(* CODESYS project TrigaPLC.project
   Title: TrigaPLC
   Author: Thalles Campagnani
   Version: 0.0.1

Project tree, tasks and I/O mapping:
  TrigaPLC : TM251MESE, Schneider Electric, order no. TM251MESE, version 4.0.6.18
      settings: OPCUA enable = True; Dummy int param for online change = 28
    application Application
      libraries: Toolbox, 2.2.0.0 (Schneider Electric); SysTimeRtc, 3.5.1.0 (System); SysTimeCore, 3.4.1.20 (System); Standard64, * (System)
      task MAST (cyclic, interval 20 ms, priority 15, watchdog 100 ms x 1) calls _001_Geral_DateAndHour
      global variables GVL
      data type Manegement
      global variables PersistentVars
      OPCUASymbolConfiguration
      data type User
      data type Group
      Symbols
      program _001_Geral_DateAndHour [CFC]
      DataLogManager
        LogFile
      trace Trace (task MAST): 
    Serial_Line_1 : Serial line, Schneider Electric, version 4.0.6.18
    Ethernet_1 : Ethernet Network, Schneider Electric, version 4.0.6.18
        settings: IPAddress = [192, 168, 1, 1]; SubnetMask = [255, 255, 255, 0]; DeviceName = 'TrigaPLC'; WebServer = TRUE; FTP Server = TRUE; SoMachine Protocol = TRUE; Modbus Server = TRUE; NetManage Protocol = TRUE; SNMP protocol = TRUE; Enable Routing = FALSE; WebVisu protocol = TRUE
    COM_Bus : COM bus, Schneider Electric, version 4.0.6.18
    IO_Bus : IO bus - TM3, Schneider Electric, version 4.0.6.18
      Module_A2 : TM3AI8/G, Schneider Electric, order no. TM3AI8/G, version 1.0.0.17
          settings: KPI Configuration.KPI Configuration[0] = 32; KPI Configuration.KPI Configuration[1] = 32; KPI Configuration.KPI Configuration[2] = 32; KPI Configuration.KPI Configuration[3] = 32; KPI Configuration.KPI Configuration[4] = 32; KPI Configuration.KPI Configuration[5] = 32; KPI Configuration.KPI Configuration[6] = 32; KPI Configuration.KPI Configuration[7] = 32; KPI Configuration.KPI Configuration[9] = 0; KPI Configuration.KPI Configuration[11] = 0; KPI Configuration.KPI Configuration[13] = 0; KPI Configuration.KPI Configuration[15] = 0; KPI Configuration.KPI Configuration[17] = 0; KPI Configuration.KPI Configuration[19] = 0; KPI Configuration.KPI Configuration[21] = 0; KPI Configuration.KPI Configuration[23] = 0; KPI Configuration.KPI Configuration[24] = 0; KPI Configuration.KPI Configuration[25] = 32; KPI Configuration.KPI Configuration[26] = 0; KPI Configuration.KPI Configuration[27] = 32; KPI Configuration.KPI Configuration[28] = 0; KPI Configuration.KPI Configuration[29] = 32; KPI Configuration.KPI Configuration[30] = 0; KPI Configuration.KPI Configuration[31] = 32; KPI Configuration.KPI Configuration[32] = 0; KPI Configuration.KPI Configuration[33] = 32; KPI Configuration.KPI Configuration[34] = 0; KPI Configuration.KPI Configuration[35] = 32; KPI Configuration.KPI Configuration[36] = 0; KPI Configuration.KPI Configuration[37] = 32; KPI Configuration.KPI Configuration[38] = 0; KPI Configuration.KPI Configuration[39] = 32; KPI Configuration.KPI Configuration[40] = 2; KPI Configuration.KPI Configuration[42] = 2; KPI Configuration.KPI Configuration[44] = 2; KPI Configuration.KPI Configuration[46] = 2; KPI Configuration.KPI Configuration[48] = 2; KPI Configuration.KPI Configuration[50] = 2; KPI Configuration.KPI Configuration[52] = 2; KPI Configuration.KPI Configuration[54] = 2
          input  inSRadAre : INT  // IW0
          input  inSRadEntPri : INT  // IW1
          input  inSRadPoc : INT  // IW2
          input  inSRadRes : INT  // IW3
          input  inSRadSaiSec : INT  // IW4
          input  inSRadAer : INT  // IW5
          input  inReserva_AI26 : INT  // IW6
          input  inReserva_AI27 : INT  // IW7
          input  ibModule_12_IBStatusIW0 : BYTE  // IBStatusIW0
          input  ibModule_12_IBStatusIW1 : BYTE  // IBStatusIW1
          input  ibModule_12_IBStatusIW2 : BYTE  // IBStatusIW2
          input  ibModule_12_IBStatusIW3 : BYTE  // IBStatusIW3
          input  ibModule_12_IBStatusIW4 : BYTE  // IBStatusIW4
          input  ibModule_12_IBStatusIW5 : BYTE  // IBStatusIW5
          input  ibModule_12_IBStatusIW6 : BYTE  // IBStatusIW6
          input  ibModule_12_IBStatusIW7 : BYTE  // IBStatusIW7
      Module_A1 : TM3AI8/G, Schneider Electric, order no. TM3AI8/G, version 1.0.0.17
          settings: KPI Configuration.KPI Configuration[0] = 32; KPI Configuration.KPI Configuration[1] = 33; KPI Configuration.KPI Configuration[2] = 32; KPI Configuration.KPI Configuration[3] = 32; KPI Configuration.KPI Configuration[4] = 32; KPI Configuration.KPI Configuration[5] = 32; KPI Configuration.KPI Configuration[6] = 32; KPI Configuration.KPI Configuration[7] = 32; KPI Configuration.KPI Configuration[9] = 0; KPI Configuration.KPI Configuration[11] = 0; KPI Configuration.KPI Configuration[13] = 0; KPI Configuration.KPI Configuration[15] = 0; KPI Configuration.KPI Configuration[17] = 0; KPI Configuration.KPI Configuration[19] = 0; KPI Configuration.KPI Configuration[21] = 0; KPI Configuration.KPI Configuration[23] = 0; KPI Configuration.KPI Configuration[24] = 0; KPI Configuration.KPI Configuration[25] = 32; KPI Configuration.KPI Configuration[26] = 0; KPI Configuration.KPI Configuration[27] = 32; KPI Configuration.KPI Configuration[28] = 0; KPI Configuration.KPI Configuration[29] = 32; KPI Configuration.KPI Configuration[30] = 0; KPI Configuration.KPI Configuration[31] = 32; KPI Configuration.KPI Configuration[32] = 0; KPI Configuration.KPI Configuration[33] = 32; KPI Configuration.KPI Configuration[34] = 0; KPI Configuration.KPI Configuration[35] = 32; KPI Configuration.KPI Configuration[36] = 0; KPI Configuration.KPI Configuration[37] = 32; KPI Configuration.KPI Configuration[38] = 0; KPI Configuration.KPI Configuration[39] = 32; KPI Configuration.KPI Configuration[40] = 2; KPI Configuration.KPI Configuration[44] = 2; KPI Configuration.KPI Configuration[46] = 2; KPI Configuration.KPI Configuration[48] = 2; KPI Configuration.KPI Configuration[50] = 2; KPI Configuration.KPI Configuration[52] = 100; KPI Configuration.KPI Configuration[54] = 2
          input  inCPer : INT  // IW0
          input  inCLogARea : INT  // IW1
          input  inCLogALin : INT  // IW2
          input  inCLogALog : INT  // IW3
          input  inCLogAPer : INT  // IW4
          input  inCParALin : INT  // IW5
          input  inCParALog : INT  // IW6
          input  inCParAPer : INT  // IW7
          input  ibModule_11_IBStatusIW0 : BYTE  // IBStatusIW0
          input  ibModule_11_IBStatusIW1 : BYTE  // IBStatusIW1
          input  ibModule_11_IBStatusIW2 : BYTE  // IBStatusIW2
          input  ibModule_11_IBStatusIW3 : BYTE  // IBStatusIW3
          input  ibModule_11_IBStatusIW4 : BYTE  // IBStatusIW4
          input  ibModule_11_IBStatusIW5 : BYTE  // IBStatusIW5
          input  ibModule_11_IBStatusIW6 : BYTE  // IBStatusIW6
          input  ibModule_11_IBStatusIW7 : BYTE  // IBStatusIW7
      Module_A0 : TM3AI8/G, Schneider Electric, order no. TM3AI8/G, version 1.0.0.17
          settings: KPI Configuration.KPI Configuration[0] = 35; KPI Configuration.KPI Configuration[1] = 35; KPI Configuration.KPI Configuration[2] = 35; KPI Configuration.KPI Configuration[3] = 35; KPI Configuration.KPI Configuration[4] = 32; KPI Configuration.KPI Configuration[5] = 32; KPI Configuration.KPI Configuration[6] = 32; KPI Configuration.KPI Configuration[7] = 32; KPI Configuration.KPI Configuration[9] = 0; KPI Configuration.KPI Configuration[11] = 0; KPI Configuration.KPI Configuration[13] = 0; KPI Configuration.KPI Configuration[15] = 0; KPI Configuration.KPI Configuration[17] = 0; KPI Configuration.KPI Configuration[19] = 0; KPI Configuration.KPI Configuration[21] = 0; KPI Configuration.KPI Configuration[23] = 0; KPI Configuration.KPI Configuration[32] = 0; KPI Configuration.KPI Configuration[33] = 32; KPI Configuration.KPI Configuration[34] = 0; KPI Configuration.KPI Configuration[35] = 32; KPI Configuration.KPI Configuration[36] = 0; KPI Configuration.KPI Configuration[37] = 32; KPI Configuration.KPI Configuration[38] = 0; KPI Configuration.KPI Configuration[39] = 32; KPI Configuration.KPI Configuration[48] = 20; KPI Configuration.KPI Configuration[50] = 20; KPI Configuration.KPI Configuration[52] = 20
          input  inReserva_AI00 : INT  // IW0
          input  inReserva_AI01 : INT  // IW1
          input  inReserva_AI02 : INT  // IW2
          input  inReserva_AI03 : INT  // IW3
          input  inBarraReg : INT  // IW4
          input  inBarraCon : INT  // IW5
          input  inBarraSeg : INT  // IW6
          input  inCLin : INT  // IW7
          input  ibModule_13_IBStatusIW0 : BYTE  // IBStatusIW0
          input  ibModule_13_IBStatusIW1 : BYTE  // IBStatusIW1
          input  ibModule_13_IBStatusIW2 : BYTE  // IBStatusIW2
          input  ibModule_13_IBStatusIW3 : BYTE  // IBStatusIW3
          input  ibModule_13_IBStatusIW4 : BYTE  // IBStatusIW4
          input  ibModule_13_IBStatusIW5 : BYTE  // IBStatusIW5
          input  ibModule_13_IBStatusIW6 : BYTE  // IBStatusIW6
          input  ibModule_13_IBStatusIW7 : BYTE  // IBStatusIW7
      Module_A3 : TM3AI8/G, Schneider Electric, order no. TM3AI8/G, version 1.0.0.17
          settings: KPI Configuration.KPI Configuration[0] = 32; KPI Configuration.KPI Configuration[1] = 32; KPI Configuration.KPI Configuration[2] = 32; KPI Configuration.KPI Configuration[3] = 32; KPI Configuration.KPI Configuration[4] = 32; KPI Configuration.KPI Configuration[5] = 32; KPI Configuration.KPI Configuration[6] = 32; KPI Configuration.KPI Configuration[7] = 32; KPI Configuration.KPI Configuration[9] = 0; KPI Configuration.KPI Configuration[11] = 0; KPI Configuration.KPI Configuration[13] = 0; KPI Configuration.KPI Configuration[15] = 0; KPI Configuration.KPI Configuration[17] = 0; KPI Configuration.KPI Configuration[19] = 0; KPI Configuration.KPI Configuration[21] = 0; KPI Configuration.KPI Configuration[23] = 0; KPI Configuration.KPI Configuration[24] = 0; KPI Configuration.KPI Configuration[25] = 32; KPI Configuration.KPI Configuration[26] = 0; KPI Configuration.KPI Configuration[27] = 32; KPI Configuration.KPI Configuration[28] = 0; KPI Configuration.KPI Configuration[29] = 32; KPI Configuration.KPI Configuration[30] = 0; KPI Configuration.KPI Configuration[31] = 32; KPI Configuration.KPI Configuration[32] = 0; KPI Configuration.KPI Configuration[33] = 32; KPI Configuration.KPI Configuration[34] = 0; KPI Configuration.KPI Configuration[35] = 32; KPI Configuration.KPI Configuration[36] = 0; KPI Configuration.KPI Configuration[37] = 32; KPI Configuration.KPI Configuration[38] = 0; KPI Configuration.KPI Configuration[39] = 32; KPI Configuration.KPI Configuration[40] = 2; KPI Configuration.KPI Configuration[42] = 2; KPI Configuration.KPI Configuration[44] = 2; KPI Configuration.KPI Configuration[46] = 2; KPI Configuration.KPI Configuration[48] = 2; KPI Configuration.KPI Configuration[50] = 2; KPI Configuration.KPI Configuration[52] = 2; KPI Configuration.KPI Configuration[54] = 2
          input  inReserva_AI30 : INT  // IW0
          input  inReserva_AI31 : INT  // IW1
          input  inReserva_AI32 : INT  // IW2
          input  inReserva_AI33 : INT  // IW3
          input  inReserva_AI34 : INT  // IW4
          input  inReserva_AI35 : INT  // IW5
          input  inReserva_AI36 : INT  // IW6
          input  inReserva_AI37 : INT  // IW7
          input  ibModule_1_IBStatusIW0 : BYTE  // IBStatusIW0
          input  ibModule_1_IBStatusIW1 : BYTE  // IBStatusIW1
          input  ibModule_1_IBStatusIW2 : BYTE  // IBStatusIW2
          input  ibModule_1_IBStatusIW3 : BYTE  // IBStatusIW3
          input  ibModule_1_IBStatusIW4 : BYTE  // IBStatusIW4
          input  ibModule_1_IBStatusIW5 : BYTE  // IBStatusIW5
          input  ibModule_1_IBStatusIW6 : BYTE  // IBStatusIW6
          input  ibModule_1_IBStatusIW7 : BYTE  // IBStatusIW7
      Module_A4 : TM3AI8/G, Schneider Electric, order no. TM3AI8/G, version 1.0.0.17
          settings: KPI Configuration.KPI Configuration[0] = 35; KPI Configuration.KPI Configuration[1] = 35; KPI Configuration.KPI Configuration[2] = 35; KPI Configuration.KPI Configuration[3] = 35; KPI Configuration.KPI Configuration[4] = 35; KPI Configuration.KPI Configuration[5] = 35; KPI Configuration.KPI Configuration[6] = 35; KPI Configuration.KPI Configuration[7] = 35; KPI Configuration.KPI Configuration[9] = 0; KPI Configuration.KPI Configuration[11] = 0; KPI Configuration.KPI Configuration[13] = 0; KPI Configuration.KPI Configuration[15] = 0; KPI Configuration.KPI Configuration[17] = 0; KPI Configuration.KPI Configuration[19] = 0; KPI Configuration.KPI Configuration[21] = 0; KPI Configuration.KPI Configuration[23] = 0; KPI Configuration.KPI Configuration[24] = 0; KPI Configuration.KPI Configuration[25] = 32; KPI Configuration.KPI Configuration[26] = 0; KPI Configuration.KPI Configuration[27] = 32; KPI Configuration.KPI Configuration[28] = 0; KPI Configuration.KPI Configuration[29] = 32; KPI Configuration.KPI Configuration[30] = 0; KPI Configuration.KPI Configuration[31] = 32; KPI Configuration.KPI Configuration[32] = 0; KPI Configuration.KPI Configuration[33] = 32; KPI Configuration.KPI Configuration[34] = 0; KPI Configuration.KPI Configuration[35] = 32; KPI Configuration.KPI Configuration[36] = 0; KPI Configuration.KPI Configuration[37] = 32; KPI Configuration.KPI Configuration[38] = 0; KPI Configuration.KPI Configuration[39] = 32; KPI Configuration.KPI Configuration[40] = 2; KPI Configuration.KPI Configuration[42] = 2; KPI Configuration.KPI Configuration[44] = 2; KPI Configuration.KPI Configuration[46] = 2; KPI Configuration.KPI Configuration[48] = 2; KPI Configuration.KPI Configuration[50] = 2; KPI Configuration.KPI Configuration[52] = 2; KPI Configuration.KPI Configuration[54] = 2
          input  inSVasPri : INT  // IW0
          input  inReserva_AI41 : INT  // IW1
          input  inReserva_AI42 : INT  // IW2
          input  inReserva_AI43 : INT  // IW3
          input  inReserva_AI44 : INT  // IW4
          input  inReserva_AI45 : INT  // IW5
          input  inReserva_AI46 : INT  // IW6
          input  inReserva_AI47 : INT  // IW7
          input  ibModule_2_IBStatusIW0 : BYTE  // IBStatusIW0
          input  ibModule_2_IBStatusIW1 : BYTE  // IBStatusIW1
          input  ibModule_2_IBStatusIW2 : BYTE  // IBStatusIW2
          input  ibModule_2_IBStatusIW3 : BYTE  // IBStatusIW3
          input  ibModule_2_IBStatusIW4 : BYTE  // IBStatusIW4
          input  ibModule_2_IBStatusIW5 : BYTE  // IBStatusIW5
          input  ibModule_2_IBStatusIW6 : BYTE  // IBStatusIW6
          input  ibModule_2_IBStatusIW7 : BYTE  // IBStatusIW7
      Module_D0 : TM3DI16/G, Schneider Electric, order no. TM3DI16/G, version 1.0.1.4
          input  inModule_D0 : WORD  // IW0
          input  inCLinBit0 : BOOL  // IW0.I0
          input  inCLinBit1 : BOOL  // IW0.I1
          input  inCLinBit2 : BOOL  // IW0.I2
          input  inReserva_DI03 : BOOL  // IW0.I3
          input  inReserva_DI04 : BOOL  // IW0.I4
          input  inReserva_DI05 : BOOL  // IW0.I5
          input  inReserva_DI06 : BOOL  // IW0.I6
          input  inReserva_DI07 : BOOL  // IW0.I7
          input  inReserva_DI08 : BOOL  // IW0.I8
          input  inReserva_DI09 : BOOL  // IW0.I9
          input  inReserva_DI010 : BOOL  // IW0.I10
          input  inReserva_DI011 : BOOL  // IW0.I11
          input  inReserva_DI012 : BOOL  // IW0.I12
          input  inReserva_DI013 : BOOL  // IW0.I13
          input  inReserva_DI014 : BOOL  // IW0.I14
          input  inReserva_DI015 : BOOL  // IW0.I15
    Ethernet_2 : Device Network, Schneider Electric, version 4.0.6.18
        settings: IPAddress = [192, 168, 2, 2]; SubnetMask = [255, 255, 255, 0]; DeviceName = 'TrigaPLC'; WebServer = TRUE; FTP Server = TRUE; SoMachine Protocol = TRUE; Modbus Server = TRUE; NetManage Protocol = TRUE; SNMP protocol = TRUE; Enable Routing = FALSE; WebVisu protocol = TRUE; DHCP Server Active = FALSE
  FdtConnections : Conexões FDT, Schneider Electric, version 1.0.0.2
  global variables GVL
*)

// TrigaPLC/Application/Manegement
TYPE Manegement :
STRUCT
 Data: User;
 DataG: Group;
 Edit: BOOL;
 New: BOOL;
 Save: BOOL;
 Delete: BOOL;
 ID: INT;
 FullAcess: BOOL;
 NullAcess: BOOL;
END_STRUCT
END_TYPE

// TrigaPLC/Application/User
TYPE User:
STRUCT
	Name: STRING[20];
	Badge: STRING[10];
	Password: STRING[8];
	Group: INT;
	Unauthorized: BOOL;
END_STRUCT
END_TYPE

// TrigaPLC/Application/Group
TYPE Group :
STRUCT
 	Access: ARRAY[0..29] OF SINT;
END_STRUCT
END_TYPE

// TrigaPLC/Application/GVL
VAR_GLOBAL
	LastUser: INT;
	LastGroup: INT;	
	Index: ARRAY[0..5] OF INT;
	Active: User;
	UserManegement: Manegement;
	DataUser: ARRAY[0..10] OF User;
	DataGroup: ARRAY [0..10] OF Group;
	UserLogin: User;
END_VAR

// TrigaPLC/Application/PersistentVars
VAR_GLOBAL PERSISTENT RETAIN

END_VAR

// GVL
VAR_GLOBAL
END_VAR

// TrigaPLC/Application/_001_Geral_DateAndHour
PROGRAM _001_Geral_DateAndHour
VAR

stGetDate: SysTimeRtc.RTS_SYSTIMEDATE;
uiGetYear: UINT;
uiGetMonth: UINT;
uiGetDay: UINT;
uiGetHour: UINT;
uiGetMinute: UINT;
uiGetSecond: UINT;
uiGetMSecond: UINT;
uiGetDayOfWeek: UINT;
uiGetYday: UINT;
uidResultConvertToDate: UDINT; 
uidResultRtcGet: UDINT;

uiSetYear: UINT;
uiSetMonth: UINT;
uiSetDay: UINT;
uiSetHour: UINT;
uiSetMinute: UINT;
uiSetSecond: UINT;
uiSetMSecond: UINT;
udiResultConvertToUtc: UDINT;
dwSetTimeStamp: DWORD;
xCommandSetRtc: BOOL;
uidResultRtcSet: UDINT;
END_VAR
VAR // added by the converter: edge detectors and wires of the graphical bodies
    _s1 : RTS_SYSTIMEDATE;
    _w1, _w4 : ANY;
    _w2 : UDINT;
    _w3 : BOOL;
END_VAR

_w1 := SysTimeRtcGet(pResult := uidResultRtcGet);
IF uidResultRtcGet = 16#0 THEN SysTimeRtcConvertUtcToDate(dwTimestampUtc := _w1, pDate := stGetDate); END_IF
uiGetYear := stGetDate.RTS_SYSTIMEDATE;
uiGetMonth := stGetDate.wYear;
uiGetDay := stGetDate.wMonth;
uiGetHour := stGetDate.wDay;
uiGetMinute := stGetDate.wHour;
uiGetSecond := stGetDate.wMinute;
uiGetMSecond := stGetDate.wSecond;
uiGetDayOfWeek := stGetDate.wMilliseconds;
uiGetYday := stGetDate.wDayOfWeek;
// compose _s1 : RTS_SYSTIMEDATE
_s1.wYear := uiSetYear;
_s1.wMonth := uiSetMonth;
_s1.wDay := uiSetDay;
_s1.wHour := uiSetHour;
_s1.wMinute := uiSetMinute;
_s1.wSecond := uiSetSecond;
_s1.wMilliseconds := uiSetMSecond;
udiResultConvertToUtc := _w2;
_w2 := SysTimeRtcConvertDateToUtc(pDate := _s1, pdwTimestampUtc := dwSetTimeStamp);
IF _w3 THEN _w4 := SysTimeRtcSet(ulTimestamp := dwSetTimeStamp); END_IF
_w3 := xCommandSetRtc AND udiResultConvertToUtc = 0;
uidResultRtcSet := _w4;

END_PROGRAM
